% RSLogix 500 project I2P HANDS-ON FINAL_BAK017.RSS, saved by version 10.00.00.00 %
PROJECT "UNTITLED"    % processor: Bul.1763 MicroLogix 1100 Series B %

PROGRAM FILES
  LAD 2 "MAIN"  10 rungs
  LAD 3 "SIM"  12 rungs
  LAD 4 "MTR"  5 rungs  % ESTOP/Stop/Start Motor %
  LAD 5   2 rungs

DATA FILES
  O0 OUTPUT  4 elements
  I1 INPUT  6 elements
  S2 STATUS  66 elements
  B3 BINARY  12 elements
  T4 TIMER  14 elements
  C5 COUNTER  1 elements
  R6 CONTROL  1 elements
  N7 INTEGER  1 elements
  F8 FLOAT  1 elements

LADDER 2 "MAIN"
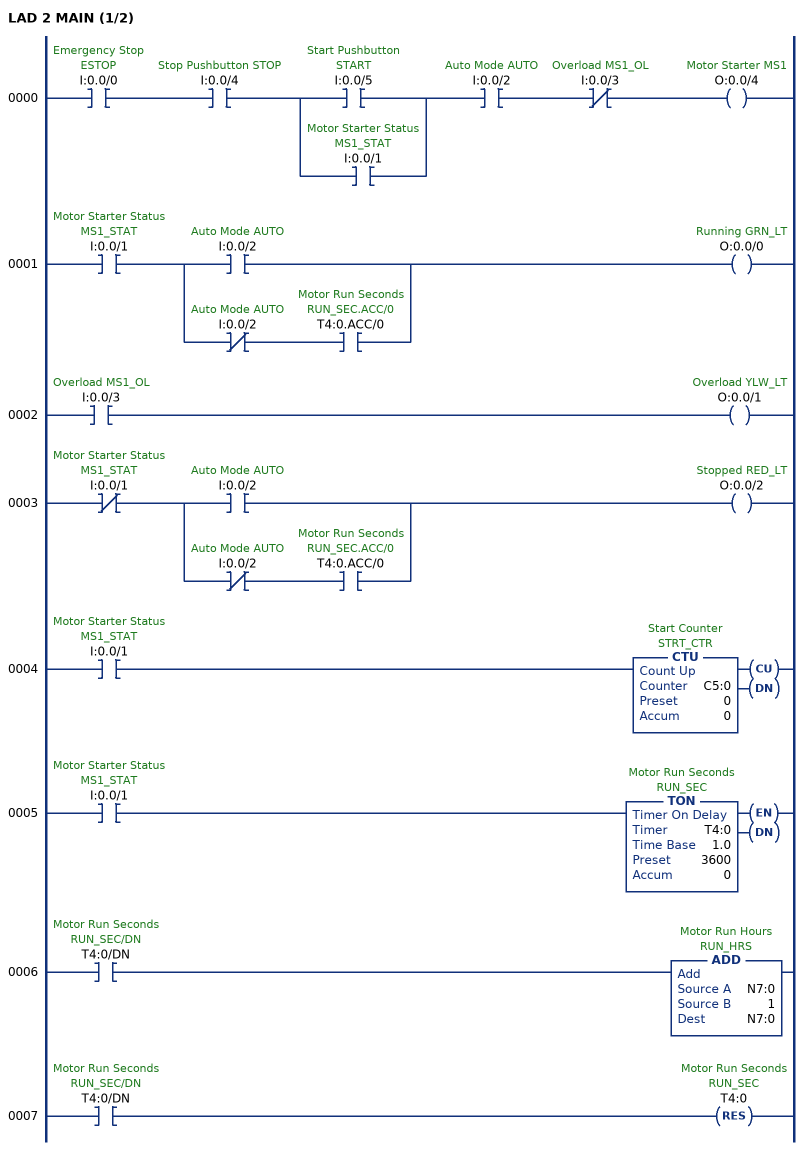
% Rung: 0 %
SOR XIC I:0.0/0 XIC I:0.0/4 BST XIC I:0.0/5 NXB XIC I:0.0/1 BND XIC I:0.0/2 XIO I:0.0/3 OTE O:0.0/4 EOR
%   I:0.0/0  ESTOP  "Emergency Stop" %
%   I:0.0/4  STOP  "Stop Pushbutton" %
%   I:0.0/5  START  "Start Pushbutton" %
%   I:0.0/1  MS1_STAT  "Motor Starter Status" %
%   I:0.0/2  AUTO  "Auto Mode" %
%   I:0.0/3  MS1_OL  "Overload" %
%   O:0.0/4  MS1  "Motor Starter" %
% Rung: 1 %
SOR XIC I:0.0/1 BST XIC I:0.0/2 NXB XIO I:0.0/2 XIC T4:0.ACC/0 BND OTE O:0.0/0 EOR
%   I:0.0/1  MS1_STAT  "Motor Starter Status" %
%   I:0.0/2  AUTO  "Auto Mode" %
%   T4:0  RUN_SEC  "Motor Run Seconds" %
%   O:0.0/0  GRN_LT  "Running" %
% Rung: 2 %
SOR XIC I:0.0/3 OTE O:0.0/1 EOR
%   I:0.0/3  MS1_OL  "Overload" %
%   O:0.0/1  YLW_LT  "Overload" %
% Rung: 3 %
SOR XIO I:0.0/1 BST XIC I:0.0/2 NXB XIO I:0.0/2 XIC T4:0.ACC/0 BND OTE O:0.0/2 EOR
%   I:0.0/1  MS1_STAT  "Motor Starter Status" %
%   I:0.0/2  AUTO  "Auto Mode" %
%   T4:0  RUN_SEC  "Motor Run Seconds" %
%   O:0.0/2  RED_LT  "Stopped" %
% Rung: 4 %
SOR XIC I:0.0/1 CTU C5:0 0 0 EOR
%   I:0.0/1  MS1_STAT  "Motor Starter Status" %
%   C5:0  STRT_CTR  "Start Counter" %
% Rung: 5 %
SOR XIC I:0.0/1 TON T4:0 1.0 3600 0 EOR
%   I:0.0/1  MS1_STAT  "Motor Starter Status" %
%   T4:0  RUN_SEC  "Motor Run Seconds" %
% Rung: 6 %
SOR XIC T4:0/DN ADD N7:0 1 N7:0 EOR
%   T4:0  RUN_SEC  "Motor Run Seconds" %
%   N7:0  RUN_HRS  "Motor Run Hours" %
% Rung: 7 %
SOR XIC T4:0/DN RES T4:0 EOR
%   T4:0  RUN_SEC  "Motor Run Seconds" %

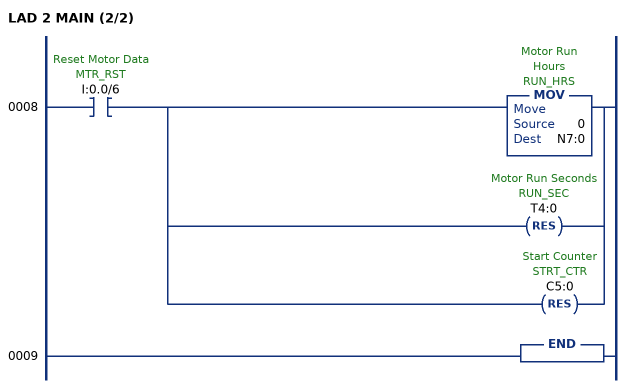
% Rung: 8 %
SOR XIC I:0.0/6 BST MOV 0 N7:0 NXB RES T4:0 NXB RES C5:0 BND EOR
%   I:0.0/6  MTR_RST  "Reset Motor Data" %
%   N7:0  RUN_HRS  "Motor Run Hours" %
%   T4:0  RUN_SEC  "Motor Run Seconds" %
%   C5:0  STRT_CTR  "Start Counter" %
% Rung: 9 %
SOR END EOR

LADDER 3 "SIM"
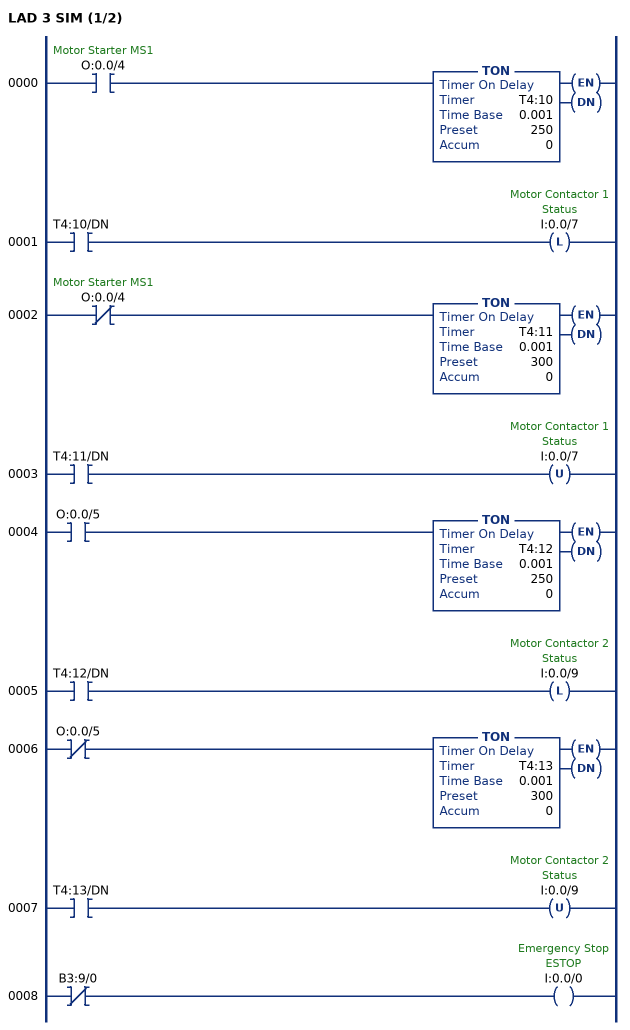
% Rung: 0 %
SOR XIC O:0.0/4 TON T4:10 0.001 250 0 EOR
%   O:0.0/4  MS1  "Motor Starter" %
% Rung: 1 %
SOR XIC T4:10/DN OTL I:0.0/7 EOR
%   I:0.0/7  "Motor Contactor 1 Status" %
% Rung: 2 %
SOR XIO O:0.0/4 TON T4:11 0.001 300 0 EOR
%   O:0.0/4  MS1  "Motor Starter" %
% Rung: 3 %
SOR XIC T4:11/DN OTU I:0.0/7 EOR
%   I:0.0/7  "Motor Contactor 1 Status" %
% Rung: 4 %
SOR XIC O:0.0/5 TON T4:12 0.001 250 0 EOR
% Rung: 5 %
SOR XIC T4:12/DN OTL I:0.0/9 EOR
%   I:0.0/9  "Motor Contactor 2 Status" %
% Rung: 6 %
SOR XIO O:0.0/5 TON T4:13 0.001 300 0 EOR
% Rung: 7 %
SOR XIC T4:13/DN OTU I:0.0/9 EOR
%   I:0.0/9  "Motor Contactor 2 Status" %
% Rung: 8 %
SOR XIO B3:9/0 OTE I:0.0/0 EOR
%   I:0.0/0  ESTOP  "Emergency Stop" %

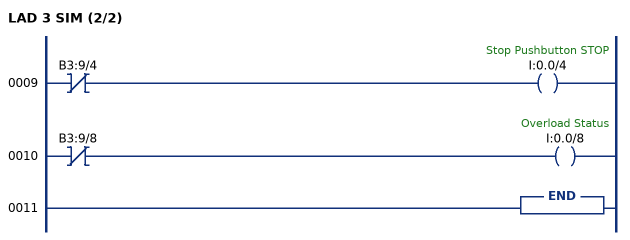
% Rung: 9 %
SOR XIO B3:9/4 OTE I:0.0/4 EOR
%   I:0.0/4  STOP  "Stop Pushbutton" %
% Rung: 10 %
SOR XIO B3:9/8 OTE I:0.0/8 EOR
%   I:0.0/8  "Overload Status" %
% Rung: 11 %
SOR END EOR

LADDER 4 "MTR"    % ESTOP/Stop/Start Motor %
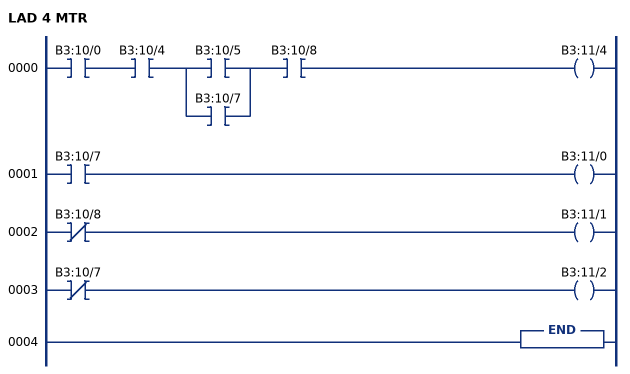
% Rung: 0 %
SOR XIC B3:10/0 XIC B3:10/4 BST XIC B3:10/5 NXB XIC B3:10/7 BND XIC B3:10/8 OTE B3:11/4 EOR
% Rung: 1 %
SOR XIC B3:10/7 OTE B3:11/0 EOR
% Rung: 2 %
SOR XIO B3:10/8 OTE B3:11/1 EOR
% Rung: 3 %
SOR XIO B3:10/7 OTE B3:11/2 EOR
% Rung: 4 %
SOR END EOR

LADDER 5
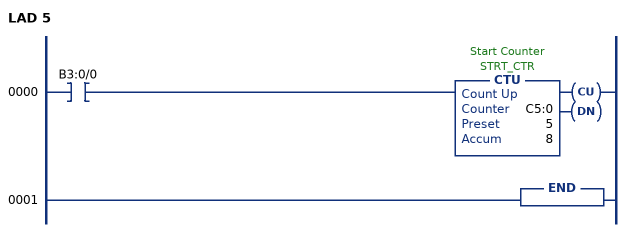
% Rung: 0 %
SOR XIC B3:0/0 CTU C5:0 5 8 EOR
%   C5:0  STRT_CTR  "Start Counter" %
% Rung: 1 %
SOR END EOR

OTHER DOCUMENTED ADDRESSES
  U:4  MTR

DATA TABLE (non-zero values as saved)
DATA B3
% B3:0 % 0X0001 0X0000 0X0000 0X0000 0X0000 0X0000 0X0000 0X0000 0X0000 0X0000
% B3:10 % 0X01A1 0X0000
DATA T4
% .PRE .ACC %
% T4:0 % 3600 0
% T4:10 % 250 0
% T4:11 % 300 0
% T4:12 % 250 0
% T4:13 % 300 0
